// TIA Portal V20 export
TYPE "udt_Andon"
   STRUCT
      inpResetReq : Bool;
      inpPressFixedStop : Bool;
      inpPressTempStop { ExternalAccessible := 'False'; ExternalVisible := 'False'; ExternalWritable := 'False'} : Bool;
      inpTAE_StopRequestReset : Bool;
      inpTAE_FixedStop : Bool;
      inpTAE_TempStop : Bool;
      inpTAE_EOT_Reached : Bool;
      outFixedStop { ExternalAccessible := 'False'; ExternalVisible := 'False'; ExternalWritable := 'False'} : Bool;   // HW interface to the physical press button lamp / HW 接口 到 physical press 按钮 lamp
      outTempStop { ExternalAccessible := 'False'; ExternalVisible := 'False'; ExternalWritable := 'False'} : Bool;   // HW interface to the physical press button lamp / HW 接口 到 physical press 按钮 lamp
      Status : Int;
   END_STRUCT;
END_TYPE
